FUNCTION_BLOCK PneumaticInsertion EXTENDS Insertion
VAR
	slider : TeknicEIP;
	screw : AirPiston;
END_VAR

slider(
	bEnable:= enable, 
	home=> , 
	outerLimit=> , 
	innerLimit=> , 
	done=> , 
	homeSet=> , 
	busy=> , 
	error=> , 
	position=> sliderPos);
	
screw(
	bEnable:= enable, 
	valveExtend=> , 
	valveRetract=> , 
	contact=> , 
	home=> , 
	innerLimit=> , 
	ready=> , 
	busy=> , 
	error=> , 
	homeSet=> );
	
home := screw.home AND slider.home;
busy := slider.busy OR screw.busy;
error := slider.error OR screw.error;

METHOD align : BOOL
VAR_INPUT
	targetPos : REAL;
END_VAR
align := slider.moveAbsolute(targetPos := targetPos);
END_METHOD

METHOD homingSequence : BOOL
IF NOT screw.homeSet THEN
	screw.homingSequence();
END_IF

IF NOT slider.homeSet THEN
	slider.homingSequence();
END_IF

homingSequence := screw.homeSet AND slider.homeSet;
END_METHOD

METHOD press : BOOL
screw.extend();
END_METHOD

METHOD release : BOOL
VAR_INPUT
END_VAR
screw.retract();
END_METHOD

METHOD traverse : BOOL
VAR_INPUT
	direction : MC_Direction;
END_VAR
slider.moveContinuous(direction := direction);
END_METHOD

END_FUNCTION_BLOCK

(* stored: Version 1.1.0.1, ProductVersion 3.1.4024.11
   POU PneumaticInsertion: Id {00f63ae2-8099-4ac0-8ac0-667b5928a006}, SpecialFunc None
   Method align: Id {e0f37983-2710-4f6f-9a4d-1bee93ed1acc}
   Method homingSequence: Id {3cd7ecee-d043-4c55-bba2-a9495d539267}
   Method press: Id {192a86da-bf4b-444b-b97f-516d139a6527}
   Method release: Id {73d5c0ca-45d8-4707-919f-ee28c6e11785}
   Method traverse: Id {bb384519-1c1e-4a43-83f9-a1cda8341fdb} *)
